{attribute addProperty BoxType "ER1018-0001-0018"}
{attribute addProperty Id "ChannelAT %I*ARRAY[0..7] OF Channel_E4AEF59E6480WcStateAT %I*WcState_F855686C1620InfoDataAT %I*InfoData_192954DE1620"}
{attribute addProperty CRC "736762842"}
{attribute addProperty SizeInBites "96"}
{attribute addProperty SizeInBytes "12"}
TYPE ER1018_C6161DDF :
STRUCT
	{attribute addProperty Name "Channel"}
	Channel : ARRAY[0..7] OF Channel_E4AEF59E;
	{attribute addProperty Name "WcState"}
	WcState : WcState_F855686C;
	{attribute addProperty Name "InfoData"}
	InfoData : InfoData_192954DE;
END_STRUCT
END_TYPE

(* stored: Version 1.2.0.0, ProductVersion 3.1.4024.9
   DUT ER1018_C6161DDF: Id {11547b2e-c187-49ea-a450-dc6e100882f0} *)
